{attribute 'qualified_only'}
{attribute 'strict'}
TYPE E_DeleteFilesByDateState :
(
	START,
	GET_FILE,
	WAIT_FOR_DELETE
);
END_TYPE

(* stored: Version 1.1.0.1, ProductVersion 3.1.4024.14
   DUT E_DeleteFilesByDateState: Id {ab0f82b1-57f4-0f6f-04f3-09fe1ce0c689} *)
